// TwinCAT 3 PLC project PlcIotMqttSampleAwsIoT
// ProgramVersion: 3.1.4021.2
// libraries:
//   Tc2_Standard, * (Beckhoff Automation GmbH)
//   Tc2_System, * (Beckhoff Automation GmbH)
//   Tc2_Utilities, * (Beckhoff Automation GmbH)
//   Tc3_IotBase, * (Beckhoff Automation GmbH)
//   Tc3_Module, * (Beckhoff Automation GmbH)
// project tree:
//   / PlcTask.TcTTO (not stored)
//   POUs/ MAIN.TcPOU, PrgMqttCom.TcPOU
// real-time tasks:
//   TASK PlcTask: cycle T#10ms, priority 20, ADS port 350

// ---- POUs/MAIN.TcPOU
PROGRAM MAIN
VAR
	m : INT;
END_VAR

m := m + 1;
PrgMqttCom();

END_PROGRAM

// ---- POUs/PrgMqttCom.TcPOU
PROGRAM PrgMqttCom
VAR
	fbMqttClient : FB_IotMqttClient;
	bSetParameter : BOOL := TRUE;
	bConnect : BOOL := TRUE;
	
	(* published message *)
	sTopicPub : STRING(255) := 'things/CX-12345';
	sPayloadPub : STRING(255);
	i: UDINT;
	fbTimer : TON := (PT:=T#1S);
	
	(* topic subscribtion *)
	bSubscribed : BOOL;
	sTopicSub : STRING(255) := 'things/CX-12345';

	(* received message *)	
	{attribute 'TcEncoding':='UTF-8'}
	sTopicRcv : STRING(255);
	{attribute 'TcEncoding':='UTF-8'}
	sPayloadRcv : STRING(255);
	
	fbMessageQueue : FB_IotMqttMessageQueue;
	fbMessage : FB_IotMqttMessage;
	
	hrErrorOccurred : HRESULT; // contains the latest occurred error
END_VAR

IF bSetParameter THEN
	bSetParameter := FALSE;
	
	(* TLS settings for AWS IoT connection *)
	fbMqttClient.stTLS.sCA := 'c:\TwinCAT\3.1\Config\Certificates\root.pem';
    fbMqttClient.stTLS.sCert := 'c:\TwinCAT\3.1\Config\Certificates\7613eee18a-certificate.pem.crt';
    fbMqttClient.stTLS.sKeyFile := 'c:\TwinCAT\3.1\Config\Certificates\7613eee18a-private.pem.key';
	
	(* Broker settings für AWS IoT *)
	fbMqttClient.sHostName:= 'a35rjvy201xp77.iot.eu-west-1.amazonaws.com';
	fbMqttClient.nHostPort:= 8883;
	fbMqttClient.sClientId:= 'CX-12345'; 
	fbMqttClient.sTopicPrefix:= ''; 
	
	fbMqttClient.ipMessageQueue := fbMessageQueue;
END_IF

fbMqttClient.Execute(bConnect);
IF fbMqttClient.bError THEN
	// add your error logging here
	hrErrorOccurred := fbMqttClient.hrErrorCode;
END_IF
IF fbMessageQueue.nQueuedMessages > 0 THEN
	IF fbMessageQueue.Dequeue(fbMessage:=fbMessage) THEN
		fbMessage.GetTopic(pTopic:=ADR(sTopicRcv), nTopicSize:=SIZEOF(sTopicRcv) );
		fbMessage.GetPayload(pPayload:=ADR(sPayloadRcv), nPayloadSize:=SIZEOF(sPayloadRcv), bSetNullTermination:=FALSE);
	END_IF
END_IF

IF fbMqttClient.bConnected THEN
	IF NOT bSubscribed THEN
		bSubscribed := fbMqttClient.Subscribe(sTopic:=sTopicSub, eQoS:=TcIotMqttQos.AtMostOnceDelivery);
		IF fbMqttClient.bError THEN
			// add your error logging here
			hrErrorOccurred := fbMqttClient.hrErrorCode;
		END_IF
	END_IF
	fbTimer(IN:=TRUE);
	IF fbTimer.Q THEN // publish new payload every second
		fbTimer(IN:=FALSE);
		i := i + 1;
		sPayloadPub := CONCAT('MyMessage', TO_STRING(i));
		fbMqttClient.Publish(	sTopic:= sTopicPub, 
								pPayload:= ADR(sPayloadPub), nPayloadSize:= LEN2(ADR(sPayloadPub)), 
								eQoS:= TcIotMqttQos.AtMostOnceDelivery, bRetain:= FALSE, bQueue:= FALSE );
		IF fbMqttClient.bError THEN
			// add your error logging here			
			hrErrorOccurred := fbMqttClient.hrErrorCode;
		END_IF
	END_IF
END_IF

END_PROGRAM
